FUNCTION_BLOCK IAS_Skill_Full (* Composite Function Block Type *)
  (* Standard: 61499-2 *)
  (* Version 0.0, 2018-04-30, 4DIAC-IDE, 4DIAC-Consortium *)
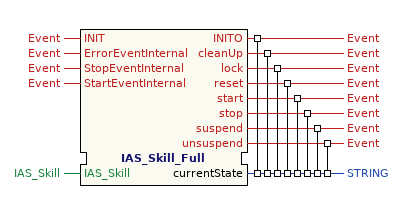
  EVENT_INPUT
    INIT; (* Initialization Request *)
    ErrorEventInternal;
    StopEventInternal;
    StartEventInternal;
  END_EVENT
  EVENT_OUTPUT
    INITO WITH currentState; (* Initialization Confirm *)
    cleanUp WITH currentState; (* Execution Confirmation *)
    lock WITH currentState;
    reset WITH currentState;
    start WITH currentState;
    stop WITH currentState;
    suspend WITH currentState;
    unsuspend WITH currentState;
  END_EVENT
  VAR_OUTPUT
    currentState : STRING;
  END_VAR
  SOCKETS
    IAS_Skill : IAS_Skill;
  END_SOCKETS
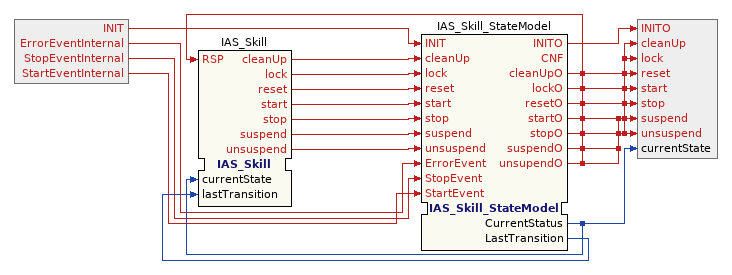
  FBS
    IAS_Skill_StateModel : IAS_Skill_StateModel;
  END_FBS
  EVENT_CONNECTIONS
    INIT TO IAS_Skill_StateModel.INIT;
    IAS_Skill.cleanUp TO IAS_Skill_StateModel.cleanUp;
    IAS_Skill.lock TO IAS_Skill_StateModel.lock;
    IAS_Skill.reset TO IAS_Skill_StateModel.reset;
    IAS_Skill.start TO IAS_Skill_StateModel.start;
    IAS_Skill.stop TO IAS_Skill_StateModel.stop;
    IAS_Skill.suspend TO IAS_Skill_StateModel.suspend;
    IAS_Skill.unsuspend TO IAS_Skill_StateModel.unsuspend;
    ErrorEventInternal TO IAS_Skill_StateModel.ErrorEvent;
    StopEventInternal TO IAS_Skill_StateModel.StopEvent;
    StartEventInternal TO IAS_Skill_StateModel.StartEvent;
    IAS_Skill_StateModel.INITO TO INITO;
    IAS_Skill_StateModel.cleanUpO TO cleanUp;
    IAS_Skill_StateModel.lockO TO lock;
    IAS_Skill_StateModel.resetO TO reset;
    IAS_Skill_StateModel.startO TO start;
    IAS_Skill_StateModel.stopO TO stop;
    IAS_Skill_StateModel.suspendO TO suspend;
    IAS_Skill_StateModel.unsupendO TO unsuspend;
    IAS_Skill_StateModel.cleanUpO TO IAS_Skill.RSP;
    IAS_Skill_StateModel.lockO TO IAS_Skill.RSP;
    IAS_Skill_StateModel.resetO TO IAS_Skill.RSP;
    IAS_Skill_StateModel.startO TO IAS_Skill.RSP;
    IAS_Skill_StateModel.stopO TO IAS_Skill.RSP;
    IAS_Skill_StateModel.suspendO TO IAS_Skill.RSP;
    IAS_Skill_StateModel.unsupendO TO IAS_Skill.RSP;
  END_CONNECTIONS
  DATA_CONNECTIONS
    IAS_Skill_StateModel.CurrentStatus TO IAS_Skill.currentState;
    IAS_Skill_StateModel.LastTransition TO IAS_Skill.lastTransition;
    IAS_Skill_StateModel.CurrentStatus TO currentState;
  END_CONNECTIONS
END_FUNCTION_BLOCK
